{attribute 'GeneratedUsingTerminal: EKM1101-0000-0016'}
{attribute addProperty BoxType "EKM1101-0000-0016"}
{attribute addProperty Id "StatusAT %I*Status_9847B4EF5"}
{attribute addProperty CRC "2915242558"}
{attribute addProperty Size "5"}
TYPE MMS_Device_Inputs_ADC3123E :
STRUCT
	{attribute addProperty Name "Status"}
	Status AT %I* : Status_9847B4EF;
END_STRUCT
END_TYPE

(* stored: Version 1.2.0.0, ProductVersion 3.1.4024.9
   DUT MMS_Device_Inputs_ADC3123E: Id {0c224d1f-9ac0-4298-abc4-74f38a0dcafb} *)
